// TIA Portal V15.1 export
// export: Created 2022-12-20T09:13:23.6419598Z, ExportSetting None, DisplayName Totally Integrated Automation Portal, DisplayVersion V15.1 Update 1, DisplayName TIA Portal Openness, DisplayVersion V15.1, DisplayName SINAMICS Startdrive Advanced, DisplayVersion V15.1, DisplayName G130, G150, S120, S150, SINAMICS MV, S210, DisplayVersion V15.1, DisplayName G110M, G120, G120C, G120D, G120P, DisplayVersion V15.1, DisplayName STEP 7 Professional, DisplayVersion V15.1 Update 1, DisplayName STEP 7 Safety, DisplayVersion V15.1, DisplayName WinCC Professional, DisplayVersion V15.1 Update 1, DisplayName SIMATIC Visualization Architect, DisplayVersion V15.1
FUNCTION_BLOCK "PLC_FB"   // FB510, FBD
TITLE = PLC FB
{ S7_Optimized_Access := 'TRUE' }
// The block is used to control the PLC and all its associated FBs and CMs
// stored: AutoNumber false, MemoryReserve 100, SetENOAutomatically false
   VAR
      Mode : "Mode_PLC_FB";   // Mode
      "000-AK01" : "CM_Cabinet_FB";   // 000-AK01
      "000-AK02" : "CM_Cabinet_FB";   // 000-AK02
      "000-AK03" : "CM_Cabinet_FB";   // 000-AK03
      "000-AS01" : "CM_Main_Panel_Control_FB";   // 000-AS01
      Energy_Save : "EnergySave";   // Energy save function block
   END_VAR
BEGIN

REGION Network 1: Call PLC mode
   // call mode block on PLC level
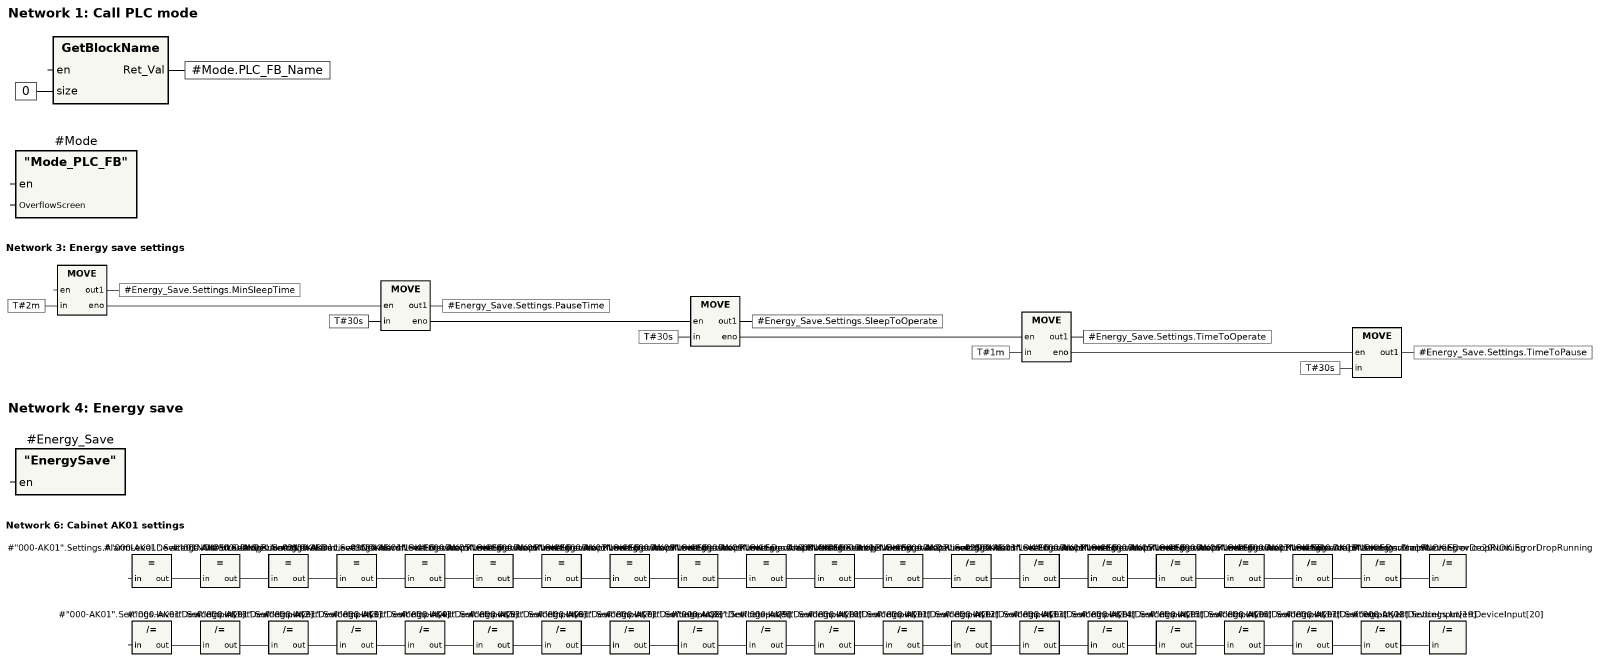
   #Mode.PLC_FB_Name := GetBlockName(size := 0);
   #Mode();   // "Mode_PLC_FB"
END_REGION

REGION Network 2: ***Energy save***
END_REGION

REGION Network 3: Energy save settings
   // Settings for energy saving
   #Energy_Save.Settings.MinSleepTime := T#2m;
   #Energy_Save.Settings.PauseTime := T#30s;
   #Energy_Save.Settings.SleepToOperate := T#30s;
   #Energy_Save.Settings.TimeToOperate := T#1m;
   #Energy_Save.Settings.TimeToPause := T#30s;
END_REGION

REGION Network 4: Energy save
   // Energy saving for whole system; triggered by end of production
   #Energy_Save();   // "EnergySave"
END_REGION

REGION Network 5: ***Cabinet***
END_REGION

REGION Network 6: Cabinet AK01 settings
   // Cabinet AK01 settings
   #"000-AK01".Settings.AlarmLevel.Device01NOK.ErrorDropRunning := TRUE;
   #"000-AK01".Settings.AlarmLevel.Device02NOK.Error := TRUE;
   #"000-AK01".Settings.AlarmLevel.Device03NOK.Error := TRUE;
   #"000-AK01".Settings.AlarmLevel.Device04NOK.ErrorDropRunning := TRUE;
   #"000-AK01".Settings.AlarmLevel.Device05NOK.ErrorDropRunning := TRUE;
   #"000-AK01".Settings.AlarmLevel.Device06NOK.ErrorDropRunning := TRUE;
   #"000-AK01".Settings.AlarmLevel.Device07NOK.ErrorDropRunning := TRUE;
   #"000-AK01".Settings.AlarmLevel.Device08NOK.ErrorDropRunning := TRUE;
   #"000-AK01".Settings.AlarmLevel.Device09NOK.ErrorDropRunning := TRUE;
   #"000-AK01".Settings.AlarmLevel.Device10NOK.ErrorDropRunning := TRUE;
   #"000-AK01".Settings.AlarmLevel.Device11NOK.ErrorDropRunning := TRUE;
   #"000-AK01".Settings.AlarmLevel.Device12NOK.Error := TRUE;
   #"000-AK01".Settings.AlarmLevel.Device13NOK.ErrorDropRunning := NOT TRUE;
   #"000-AK01".Settings.AlarmLevel.Device14NOK.ErrorDropRunning := NOT TRUE;
   #"000-AK01".Settings.AlarmLevel.Device15NOK.ErrorDropRunning := NOT TRUE;
   #"000-AK01".Settings.AlarmLevel.Device16NOK.ErrorDropRunning := NOT TRUE;
   #"000-AK01".Settings.AlarmLevel.Device17NOK.ErrorDropRunning := NOT TRUE;
   #"000-AK01".Settings.AlarmLevel.Device18NOK.ErrorDropRunning := NOT TRUE;
   #"000-AK01".Settings.AlarmLevel.Device19NOK.ErrorDropRunning := NOT TRUE;
   #"000-AK01".Settings.AlarmLevel.Device20NOK.ErrorDropRunning := NOT TRUE;
   #"000-AK01".Settings.InvertDeviceInput[1] := NOT TRUE;
   #"000-AK01".Settings.InvertDeviceInput[2] := NOT TRUE;
   #"000-AK01".Settings.InvertDeviceInput[3] := NOT TRUE;
   #"000-AK01".Settings.InvertDeviceInput[4] := NOT TRUE;
   #"000-AK01".Settings.InvertDeviceInput[5] := NOT TRUE;
   #"000-AK01".Settings.InvertDeviceInput[6] := NOT TRUE;
   #"000-AK01".Settings.InvertDeviceInput[7] := NOT TRUE;
   #"000-AK01".Settings.InvertDeviceInput[8] := NOT TRUE;
   #"000-AK01".Settings.InvertDeviceInput[9] := NOT TRUE;
   #"000-AK01".Settings.InvertDeviceInput[10] := NOT TRUE;
   #"000-AK01".Settings.InvertDeviceInput[11] := NOT TRUE;
   #"000-AK01".Settings.InvertDeviceInput[12] := NOT TRUE;
   #"000-AK01".Settings.InvertDeviceInput[13] := NOT TRUE;
   #"000-AK01".Settings.InvertDeviceInput[14] := NOT TRUE;
   #"000-AK01".Settings.InvertDeviceInput[15] := NOT TRUE;
   #"000-AK01".Settings.InvertDeviceInput[16] := NOT TRUE;
   #"000-AK01".Settings.InvertDeviceInput[17] := NOT TRUE;
   #"000-AK01".Settings.InvertDeviceInput[18] := NOT TRUE;
   #"000-AK01".Settings.InvertDeviceInput[19] := NOT TRUE;
   #"000-AK01".Settings.InvertDeviceInput[20] := NOT TRUE;
END_REGION

REGION Network 7: Call CM Cabinet AK01
   // Call CM Cabinet AK01
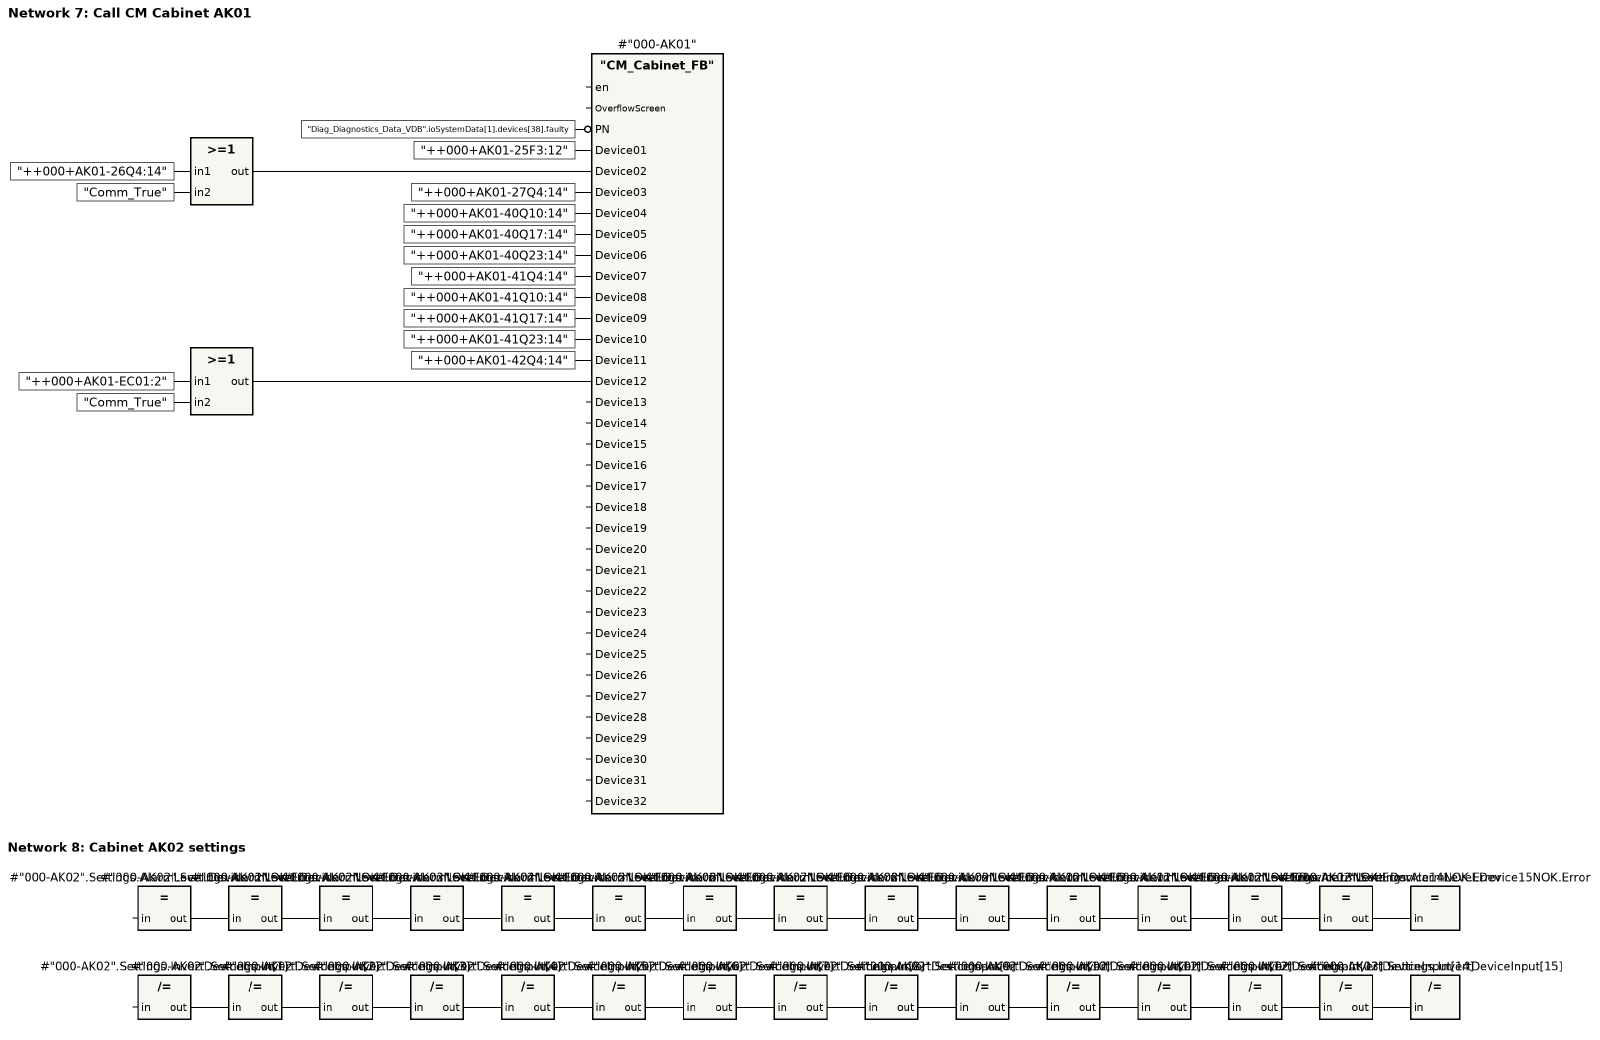
   #"000-AK01"(PN := NOT "Diag_Diagnostics_Data_VDB".ioSystemData[1].devices[38].faulty,   // "CM_Cabinet_FB"
               Device01 := "++000+AK01-25F3:12",
               Device02 := "++000+AK01-26Q4:14" OR "Comm_True",
               Device03 := "++000+AK01-27Q4:14",
               Device04 := "++000+AK01-40Q10:14",
               Device05 := "++000+AK01-40Q17:14",
               Device06 := "++000+AK01-40Q23:14",
               Device07 := "++000+AK01-41Q4:14",
               Device08 := "++000+AK01-41Q10:14",
               Device09 := "++000+AK01-41Q17:14",
               Device10 := "++000+AK01-41Q23:14",
               Device11 := "++000+AK01-42Q4:14",
               Device12 := "++000+AK01-EC01:2" OR "Comm_True");
END_REGION

REGION Network 8: Cabinet AK02 settings
   // Cabinet AK02 settings
   #"000-AK02".Settings.AlarmLevel.Device01NOK.Error := TRUE;
   #"000-AK02".Settings.AlarmLevel.Device02NOK.Error := TRUE;
   #"000-AK02".Settings.AlarmLevel.Device03NOK.Error := TRUE;
   #"000-AK02".Settings.AlarmLevel.Device04NOK.Error := TRUE;
   #"000-AK02".Settings.AlarmLevel.Device05NOK.Error := TRUE;
   #"000-AK02".Settings.AlarmLevel.Device06NOK.Error := TRUE;
   #"000-AK02".Settings.AlarmLevel.Device07NOK.Error := TRUE;
   #"000-AK02".Settings.AlarmLevel.Device08NOK.Error := TRUE;
   #"000-AK02".Settings.AlarmLevel.Device09NOK.Error := TRUE;
   #"000-AK02".Settings.AlarmLevel.Device10NOK.Error := TRUE;
   #"000-AK02".Settings.AlarmLevel.Device11NOK.Error := TRUE;
   #"000-AK02".Settings.AlarmLevel.Device12NOK.Error := TRUE;
   #"000-AK02".Settings.AlarmLevel.Device13NOK.Error := TRUE;
   #"000-AK02".Settings.AlarmLevel.Device14NOK.Error := TRUE;
   #"000-AK02".Settings.AlarmLevel.Device15NOK.Error := TRUE;
   #"000-AK02".Settings.InvertDeviceInput[1] := NOT TRUE;
   #"000-AK02".Settings.InvertDeviceInput[2] := NOT TRUE;
   #"000-AK02".Settings.InvertDeviceInput[3] := NOT TRUE;
   #"000-AK02".Settings.InvertDeviceInput[4] := NOT TRUE;
   #"000-AK02".Settings.InvertDeviceInput[5] := NOT TRUE;
   #"000-AK02".Settings.InvertDeviceInput[6] := NOT TRUE;
   #"000-AK02".Settings.InvertDeviceInput[7] := NOT TRUE;
   #"000-AK02".Settings.InvertDeviceInput[8] := NOT TRUE;
   #"000-AK02".Settings.InvertDeviceInput[9] := NOT TRUE;
   #"000-AK02".Settings.InvertDeviceInput[10] := NOT TRUE;
   #"000-AK02".Settings.InvertDeviceInput[11] := NOT TRUE;
   #"000-AK02".Settings.InvertDeviceInput[12] := NOT TRUE;
   #"000-AK02".Settings.InvertDeviceInput[13] := NOT TRUE;
   #"000-AK02".Settings.InvertDeviceInput[14] := NOT TRUE;
   #"000-AK02".Settings.InvertDeviceInput[15] := NOT TRUE;
END_REGION

REGION Network 9: Call CM Cabinet AK02
   // Call CM Cabinet AK02
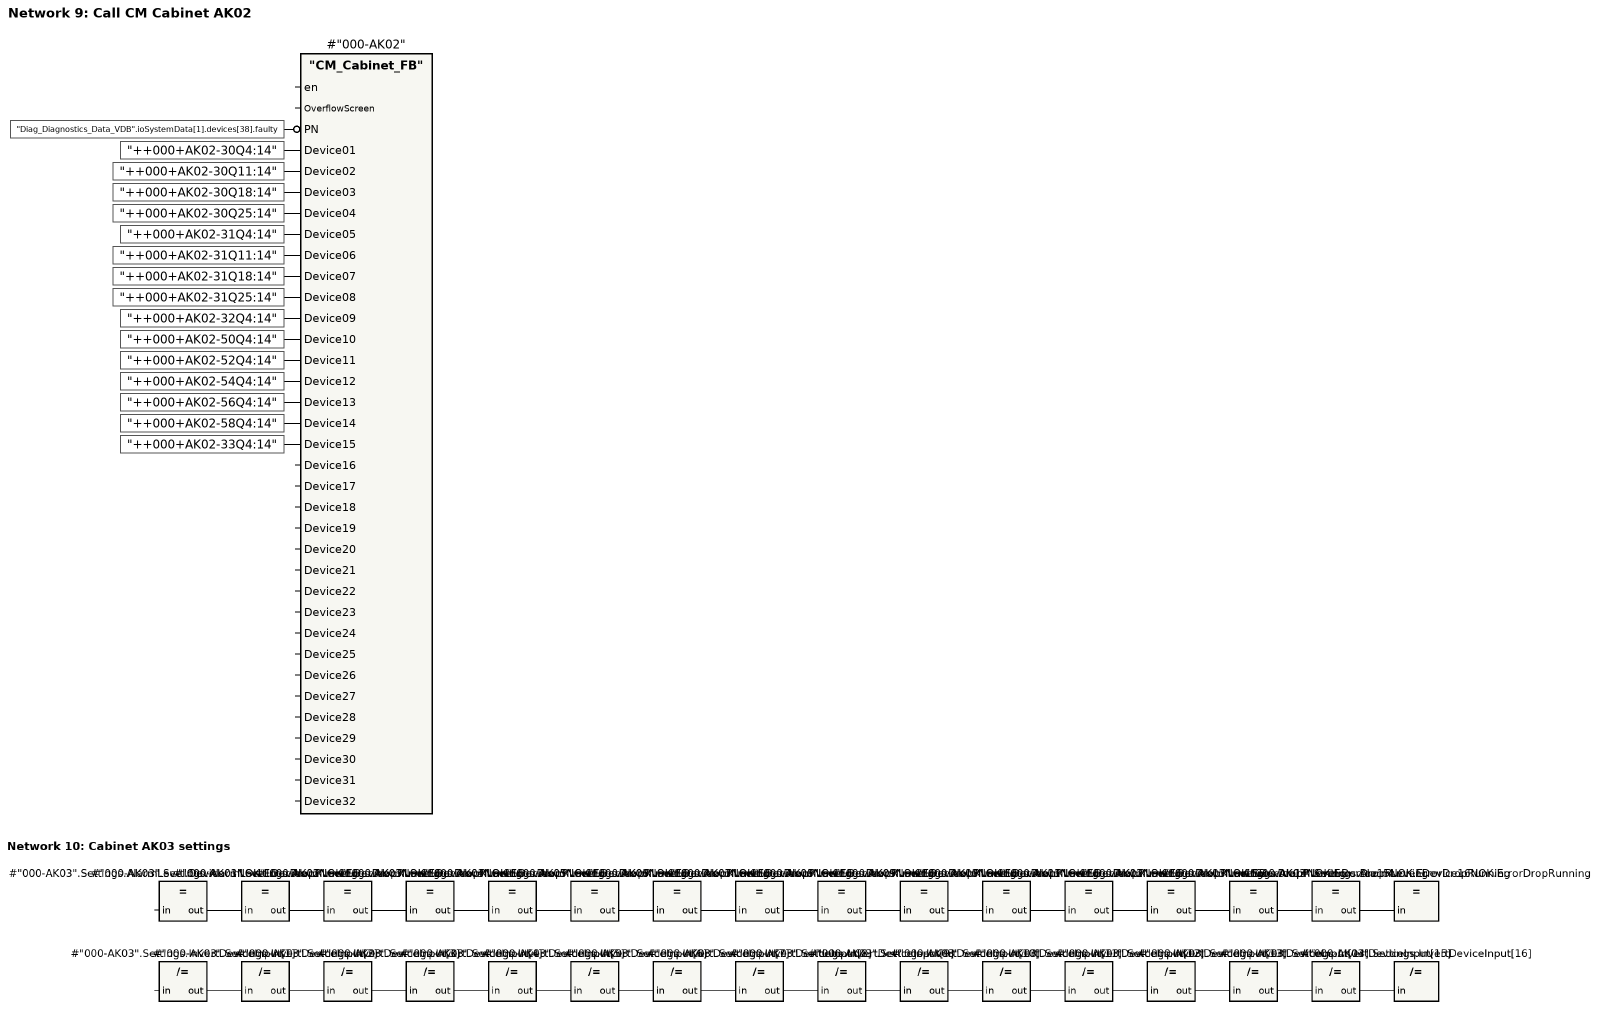
   #"000-AK02"(PN := NOT "Diag_Diagnostics_Data_VDB".ioSystemData[1].devices[38].faulty,   // "CM_Cabinet_FB"
               Device01 := "++000+AK02-30Q4:14",
               Device02 := "++000+AK02-30Q11:14",
               Device03 := "++000+AK02-30Q18:14",
               Device04 := "++000+AK02-30Q25:14",
               Device05 := "++000+AK02-31Q4:14",
               Device06 := "++000+AK02-31Q11:14",
               Device07 := "++000+AK02-31Q18:14",
               Device08 := "++000+AK02-31Q25:14",
               Device09 := "++000+AK02-32Q4:14",
               Device10 := "++000+AK02-50Q4:14",
               Device11 := "++000+AK02-52Q4:14",
               Device12 := "++000+AK02-54Q4:14",
               Device13 := "++000+AK02-56Q4:14",
               Device14 := "++000+AK02-58Q4:14",
               Device15 := "++000+AK02-33Q4:14");
END_REGION

REGION Network 10: Cabinet AK03 settings
   // Cabinet AK03 settings
   #"000-AK03".Settings.AlarmLevel.Device01NOK.ErrorDropRunning := TRUE;
   #"000-AK03".Settings.AlarmLevel.Device02NOK.ErrorDropRunning := TRUE;
   #"000-AK03".Settings.AlarmLevel.Device03NOK.ErrorDropRunning := TRUE;
   #"000-AK03".Settings.AlarmLevel.Device04NOK.ErrorDropRunning := TRUE;
   #"000-AK03".Settings.AlarmLevel.Device05NOK.ErrorDropRunning := TRUE;
   #"000-AK03".Settings.AlarmLevel.Device06NOK.ErrorDropRunning := TRUE;
   #"000-AK03".Settings.AlarmLevel.Device07NOK.ErrorDropRunning := TRUE;
   #"000-AK03".Settings.AlarmLevel.Device08NOK.ErrorDropRunning := TRUE;
   #"000-AK03".Settings.AlarmLevel.Device09NOK.ErrorDropRunning := TRUE;
   #"000-AK03".Settings.AlarmLevel.Device10NOK.ErrorDropRunning := TRUE;
   #"000-AK03".Settings.AlarmLevel.Device11NOK.ErrorDropRunning := TRUE;
   #"000-AK03".Settings.AlarmLevel.Device12NOK.ErrorDropRunning := TRUE;
   #"000-AK03".Settings.AlarmLevel.Device13NOK.ErrorDropRunning := TRUE;
   #"000-AK03".Settings.AlarmLevel.Device14NOK.ErrorDropRunning := TRUE;
   #"000-AK03".Settings.AlarmLevel.Device15NOK.ErrorDropRunning := TRUE;
   #"000-AK03".Settings.AlarmLevel.Device16NOK.ErrorDropRunning := TRUE;
   #"000-AK03".Settings.InvertDeviceInput[1] := NOT TRUE;
   #"000-AK03".Settings.InvertDeviceInput[2] := NOT TRUE;
   #"000-AK03".Settings.InvertDeviceInput[3] := NOT TRUE;
   #"000-AK03".Settings.InvertDeviceInput[4] := NOT TRUE;
   #"000-AK03".Settings.InvertDeviceInput[5] := NOT TRUE;
   #"000-AK03".Settings.InvertDeviceInput[6] := NOT TRUE;
   #"000-AK03".Settings.InvertDeviceInput[7] := NOT TRUE;
   #"000-AK03".Settings.InvertDeviceInput[8] := NOT TRUE;
   #"000-AK03".Settings.InvertDeviceInput[9] := NOT TRUE;
   #"000-AK03".Settings.InvertDeviceInput[10] := NOT TRUE;
   #"000-AK03".Settings.InvertDeviceInput[11] := NOT TRUE;
   #"000-AK03".Settings.InvertDeviceInput[12] := NOT TRUE;
   #"000-AK03".Settings.InvertDeviceInput[13] := NOT TRUE;
   #"000-AK03".Settings.InvertDeviceInput[14] := NOT TRUE;
   #"000-AK03".Settings.InvertDeviceInput[15] := NOT TRUE;
   #"000-AK03".Settings.InvertDeviceInput[16] := NOT TRUE;
END_REGION

REGION Network 11: Call CM Cabinet AK03
   // Call CM Cabinet AK03
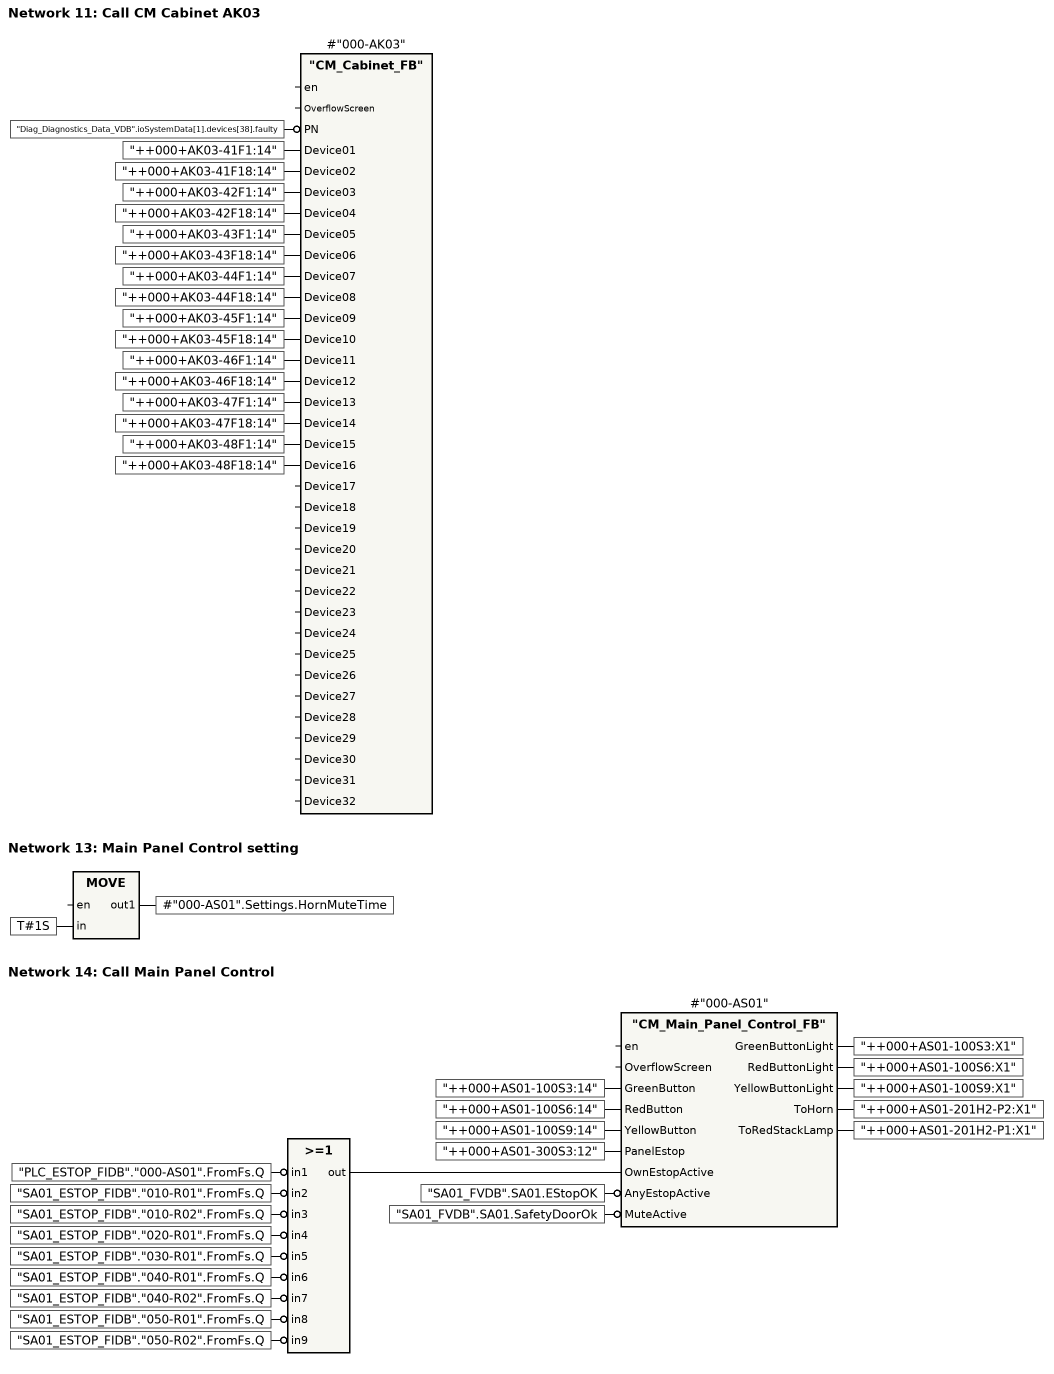
   #"000-AK03"(PN := NOT "Diag_Diagnostics_Data_VDB".ioSystemData[1].devices[38].faulty,   // "CM_Cabinet_FB"
               Device01 := "++000+AK03-41F1:14",
               Device02 := "++000+AK03-41F18:14",
               Device03 := "++000+AK03-42F1:14",
               Device04 := "++000+AK03-42F18:14",
               Device05 := "++000+AK03-43F1:14",
               Device06 := "++000+AK03-43F18:14",
               Device07 := "++000+AK03-44F1:14",
               Device08 := "++000+AK03-44F18:14",
               Device09 := "++000+AK03-45F1:14",
               Device10 := "++000+AK03-45F18:14",
               Device11 := "++000+AK03-46F1:14",
               Device12 := "++000+AK03-46F18:14",
               Device13 := "++000+AK03-47F1:14",
               Device14 := "++000+AK03-47F18:14",
               Device15 := "++000+AK03-48F1:14",
               Device16 := "++000+AK03-48F18:14");
END_REGION

REGION Network 12: *** Main control panel ***
END_REGION

REGION Network 13: Main Panel Control setting
   // Settings for:
   // - Horn muting
   #"000-AS01".Settings.HornMuteTime := T#1S;
END_REGION

REGION Network 14: Call Main Panel Control
   // 000-AS01
   #"000-AS01"(GreenButton := "++000+AS01-100S3:14",   // "CM_Main_Panel_Control_FB"
               RedButton := "++000+AS01-100S6:14",
               YellowButton := "++000+AS01-100S9:14",
               PanelEstop := "++000+AS01-300S3:12",
               OwnEstopActive := NOT "PLC_ESTOP_FIDB"."000-AS01".FromFs.Q OR NOT "SA01_ESTOP_FIDB"."010-R01".FromFs.Q OR NOT "SA01_ESTOP_FIDB"."010-R02".FromFs.Q OR NOT "SA01_ESTOP_FIDB"."020-R01".FromFs.Q OR NOT "SA01_ESTOP_FIDB"."030-R01".FromFs.Q OR NOT "SA01_ESTOP_FIDB"."040-R01".FromFs.Q OR NOT "SA01_ESTOP_FIDB"."040-R02".FromFs.Q OR NOT "SA01_ESTOP_FIDB"."050-R01".FromFs.Q OR NOT "SA01_ESTOP_FIDB"."050-R02".FromFs.Q,
               AnyEstopActive := NOT "SA01_FVDB".SA01.EStopOK,
               MuteActive := NOT "SA01_FVDB".SA01.SafetyDoorOk,
               GreenButtonLight => "++000+AS01-100S3:X1",
               RedButtonLight => "++000+AS01-100S6:X1",
               YellowButtonLight => "++000+AS01-100S9:X1",
               ToHorn => "++000+AS01-201H2-P2:X1",
               ToRedStackLamp => "++000+AS01-201H2-P1:X1");
END_REGION

REGION Network 15: *** Call structure***
END_REGION

REGION Network 16: Call system
   // Collect system data
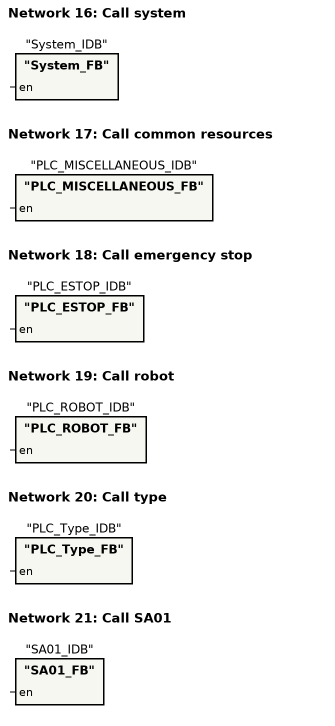
   "System_IDB"();   // "System_FB"
END_REGION

REGION Network 17: Call common resources
   // Equipment that is not linked to one SA or EM
   "PLC_MISCELLANEOUS_IDB"();   // "PLC_MISCELLANEOUS_FB"
END_REGION

REGION Network 18: Call emergency stop
   // Estops that switch off the complete line
   "PLC_ESTOP_IDB"();   // "PLC_ESTOP_FB"
END_REGION

REGION Network 19: Call robot
   // Robot functions
   "PLC_ROBOT_IDB"();   // "PLC_ROBOT_FB"
END_REGION

REGION Network 20: Call type
   // Main type fb
   "PLC_Type_IDB"();   // "PLC_Type_FB"
END_REGION

REGION Network 21: Call SA01
   // Call safety area 1
   "SA01_IDB"();   // "SA01_FB"
END_REGION
END_FUNCTION_BLOCK
